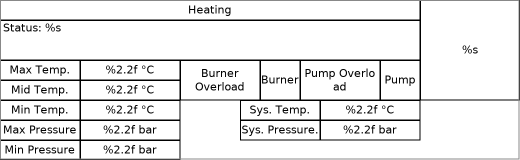
VISUALIZATION UI_Heating  // 520x160
VAR_IN_OUT
	pou			: Heating;
END_VAR
VAR
END_VAR
    Rectangle (0,0 420x20), "Heating"
    Rectangle (0,20 420x40), "Status: %s", text variable: pou._ctx.hmi.sStatusText
        p55702900: pou._ctx.hmi.nStatusColor
    Rectangle (420,0 100x100), "%s", text variable: pou._ctx.hmi.sButtonText
        p55702900: pou._ctx.hmi.nButtonColor
        toggle pou._ctx.hmi.bButton
    Rectangle (0,60 80x20), "Max Temp."
    Rectangle (0,80 80x20), "Mid Temp."
    Rectangle (0,100 80x20), "Min Temp."
    Rectangle (80,60 100x20), "%2.2f °C", text variable: pou._ctx.hmi.rMaxTemperature
        OnMouseClick: write the text variable via Default
    Rectangle (80,80 100x20), "%2.2f °C", text variable: pou._ctx.hmi.rStdTemperature
        OnMouseClick: write the text variable via Default
    Rectangle (80,100 100x20), "%2.2f °C", text variable: pou._ctx.hmi.rMinTemperature
        OnMouseClick: write the text variable via Default
    Rectangle (0,140 80x20), "Min Pressure"
    Rectangle (0,120 80x20), "Max Pressure"
    Rectangle (80,120 100x20), "%2.2f bar", text variable: pou._ctx.hmi.rMaxPressure
        OnMouseClick: write the text variable via Default
    Rectangle (80,140 100x20), "%2.2f bar", text variable: pou._ctx.hmi.rMinPressure
        OnMouseClick: write the text variable via Default
    Rectangle (380,60 40x40), "Pump", colour toggle: pou.bPump
        toggle pou.bPump
    Rectangle (260,60 40x40), "Burner", colour toggle: pou.bBurner
        toggle pou.bBurner
    Rectangle (300,60 80x40), "Pump Overload", colour toggle: pou.bPumpOverload
        toggle pou.bPumpOverload
    Rectangle (180,60 80x40), "Burner Overload", colour toggle: pou.bBurnerOverload
        toggle pou.bBurnerOverload
    Rectangle (320,120 100x20), "%2.2f bar", text variable: pou.rBoilerPressure
    Rectangle (240,100 80x20), "Sys. Temp."
    Rectangle (240,120 80x20), "Sys. Pressure."
    Rectangle (320,100 100x20), "%2.2f °C", text variable: pou.rBoilerTemp
END_VISUALIZATION

(* stored: Version 1.1.0.1
   Visu UI_Heating: Id {5e975df5-f9d8-4266-ac63-1a697bad235c} *)
